FUNCTION_BLOCK CTRL_PID (* FT_PI is a PI controller with manual functionality. *)
  (* Standard: 61499-1; Description: version 2.0	30. jun. 2008 programmer 	hugo tested by	oscat FT_PI is a PI controller with manual functionality. The PID controller works according to the fomula Y = e *(KP+ KI * INTEG(e) ) + offset, while e = set_point - actual. a rst will reset all internal data, while a switch to manual will cause the controller to follow the function Y = manual_in + offset. limit_h and Limit_l set the possible output range of Y. the output flags lim will signal that the output limits are active. *)
  (* Version 1.0, 2025-12-19, franz *)
  PACKAGE OSCAT::Basic::POUs::Engineering::Control;
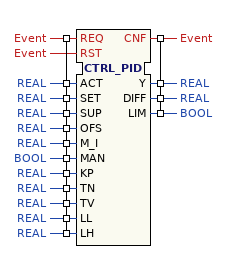
  EVENT_INPUT
    REQ WITH ACT, SET, SUP, OFS, M_I, MAN, KP, TN, TV, LL, LH; (* Normal Execution Request *)
    RST; (* Reset *)
  END_EVENT
  EVENT_OUTPUT
    CNF WITH Y, DIFF, LIM; (* Execution Confirmation *)
  END_EVENT
  VAR_INPUT
    ACT : REAL; (* Actual Value *)
    SET : REAL; (* Set Point *)
    SUP : REAL; (* Noise Suppression *)
    OFS : REAL; (* Offset *)
    M_I : REAL; (* Manual Input *)
    MAN : BOOL; (* Manual Mode *)
    KP : REAL := 1.0; (* Proportional Gain *)
    TN : REAL := 1.0; (* Integral Time *)
    TV : REAL := 1.0; (* Derivative Time *)
    LL : REAL := -1000.0; (* Limit Low *)
    LH : REAL := 1000.0; (* Limit High *)
  END_VAR
  VAR_OUTPUT
    Y : REAL; (* Output *)
    DIFF : REAL; (* Difference *)
    LIM : BOOL; (* Limit Reached *)
  END_VAR
  FBS
    pid : OSCAT::Basic::POUs::Engineering::Control::FT_PIDWL; (* Internal PID controller *)
    co : OSCAT::Basic::POUs::Engineering::Control::CTRL_OUT; (* Internal Control Output Instance *)
  END_FBS
  EC_STATES
    REQ : REQ -> CNF;
    RST : RST -> CNF;
  END_STATES
  ALGORITHM RST IN ST:
pid.RST();
  END_ALGORITHM
  ALGORITHM REQ IN ST:
DIFF := CTRL_IN(SET, ACT, SUP);

(* Call internal PID instance *)
pid.REQ(in := DIFF, kp := KP, tn := TN, tv := TV, lim_l := LL, lim_h := LH);

(* Call internal Control Output instance *)
co(ci := pid.Y, OFFSET := OFS, man_in := M_I, lim_l := LL, lim_h := LH, MANUAL := MAN);

Y := co.Y;
LIM := co.LIM;

(* Original OSCAT revision history retained for documentation hm 1.12.2006 rev 1.1 changed
 * algorithm to trapezregel hm 3.1.2007 rev 1.2 added integ_band hm 3.3.2007 rev 1.3 added
 * default values hm 31.oct 2007 rev 1.4 total rewrite hm 3.11.2007 rev 1.5 added noise input hm
 * 5. jan 2008 rev 1.6 improved code *)
  END_ALGORITHM
END_FUNCTION_BLOCK
